
FUNCTION CB_sel_dt : dt


TITLE = ' Binary selection on 2 variables '
VERSION : '1.0'
AUTHOR  : CB
NAME    : sel_dt
FAMILY  : TNI

VAR_INPUT
    G : BOOL;
    IN0 : DT ;
    IN1 : DT ;

END_VAR

BEGIN

CB_sel_dt := SEL(G:= G, IN0 := IN0, IN1 := IN1);

END_FUNCTION
